// TwinCAT 3 PLC project Main
// ProgramVersion: 3.1.4024.0
// libraries:
//   Tc2_Standard, * (Beckhoff Automation GmbH)
//   Tc2_System, * (Beckhoff Automation GmbH)
//   Tc3_Module, * (Beckhoff Automation GmbH)
// project tree:
//   / PlcTask.TcTTO
//   POUs/ CFCPOU.TcPOU, FBDPOU.TcPOU, LDPOU.TcPOU, STPOU.TcPOU
// real-time tasks:
//   TASK PlcTask: cycle T#10ms, priority 20, ADS port 350

CONFIGURATION Main
    RESOURCE PLC ON TwinCAT3
        TASK PlcTask(INTERVAL := T#10ms, PRIORITY := 20);
        PROGRAM LDPOU WITH PlcTask : LDPOU;
        PROGRAM FBDPOU WITH PlcTask : FBDPOU;
        PROGRAM CFCPOU WITH PlcTask : CFCPOU;
        PROGRAM STPOU WITH PlcTask : STPOU;
    END_RESOURCE
END_CONFIGURATION

// ---- POUs/LDPOU.TcPOU
PROGRAM LDPOU
VAR
	// Start Button
	btnStart: BOOL;
	// Stop Button
	btnStop: BOOL;
	// Motor Starter Coil
	Coil: BOOL;
END_VAR

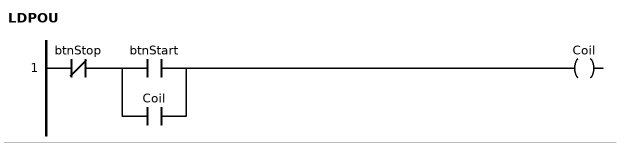
// NETWORK 1
Coil := NOT btnStop AND (btnStart OR Coil);

END_PROGRAM

// ---- POUs/FBDPOU.TcPOU
PROGRAM FBDPOU
VAR
	// Start Button
	btnStart: BOOL;
	// Stop Button
	btnStop: BOOL;
	// Motor Starter Coil
	Coil: BOOL;
END_VAR

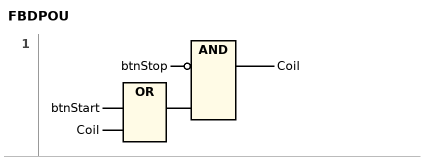
// NETWORK 1
Coil := NOT btnStop AND (btnStart OR Coil);

END_PROGRAM

// ---- POUs/CFCPOU.TcPOU
PROGRAM CFCPOU
VAR
	// Start Button
	btnStart: BOOL;
	// Stop Button
	btnStop: BOOL;
	// Motor Starter Coil
	Coil: BOOL;
END_VAR
VAR // added by the converter: edge detectors and wires of the graphical bodies
    _w1 : BOOL;
END_VAR

Coil := NOT btnStop AND _w1;
_w1 := btnStart OR Coil;

END_PROGRAM

// ---- POUs/STPOU.TcPOU
PROGRAM STPOU
VAR
	// Start Button
	btnStart: BOOL;
	// Stop Button
	btnStop: BOOL;
	// Motor Starter Coil
	Coil: BOOL;
END_VAR

Coil := NOT btnStop AND (btnStart OR Coil);

END_PROGRAM
